(* CODESYS project PruebaReporte22.project

Project tree, tasks and I/O mapping:
  Device : CECC-LK, Festo AG & Co. KG, order no. 574418, version 3.5.3.1
    application Application
      libraries: Standard, * (System)
      task MainTask (cyclic, interval t#20ms, priority 20) calls PLC_PRG
      program PLC_PRG [LD]
      visualisation Visualization
    Onboard : CECC 14I/8O, Festo AG & Co. KG, version 3.4.5.5
        unmapped channels: Onboard Input, Onboard Output
      Digital Inputs
          unmapped channels: Onboard Input
      Digital Outputs
          unmapped channels: Onboard Output
  text list GlobalTextList
*)

// Device/Application/PLC_PRG
PROGRAM PLC_PRG
VAR
	S1: BOOL;
	B1: BOOL;
	Y1: BOOL;
	S2: BOOL;
	inicio: BOOL;
	Y3: BOOL;
	Y4: BOOL;
	Y2: BOOL;
	prevB1: BOOL;
	pulso: BOOL;
	fase: BOOL;
END_VAR
VAR // added by the converter: edge detectors and wires of the graphical bodies
    _w1, _w2, _w3 : BOOL;
END_VAR

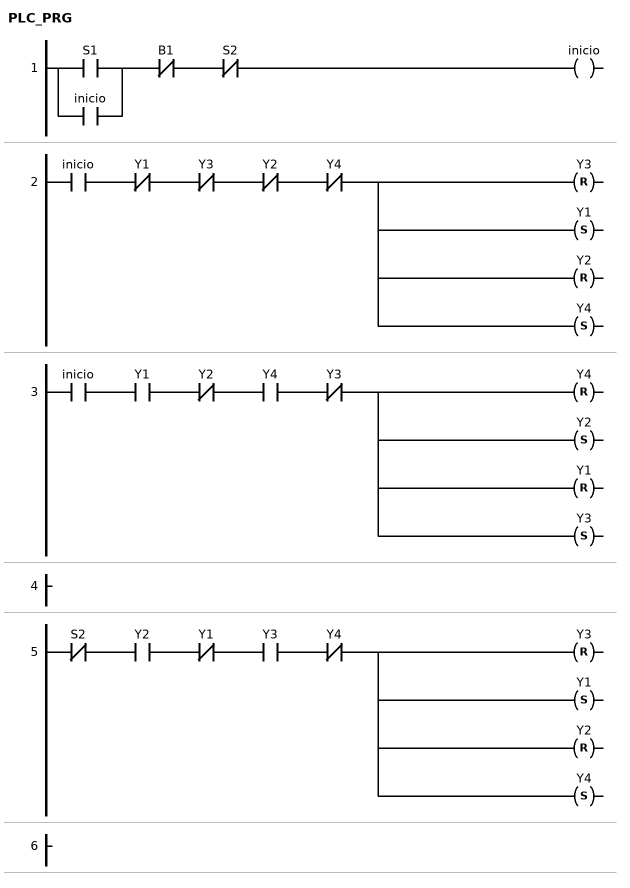
// NETWORK 1
inicio := (S1 OR inicio) AND NOT B1 AND NOT S2;

// NETWORK 2
_w1 := inicio AND NOT Y1 AND NOT Y3 AND NOT Y2 AND NOT Y4;
Y3 R= _w1;
Y1 S= _w1;
Y2 R= _w1;
Y4 S= _w1;

// NETWORK 3
_w2 := inicio AND Y1 AND NOT Y2 AND Y4 AND NOT Y3;
Y4 R= _w2;
Y2 S= _w2;
Y1 R= _w2;
Y3 S= _w2;

// NETWORK 4

// NETWORK 5
_w3 := NOT S2 AND Y2 AND NOT Y1 AND Y3 AND NOT Y4;
Y3 R= _w3;
Y1 S= _w3;
Y2 R= _w3;
Y4 S= _w3;

// NETWORK 6

END_PROGRAM

// Device/Application/Visualization
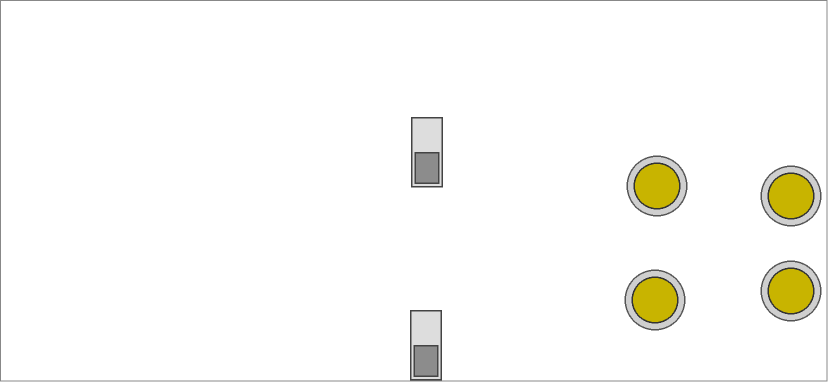
VISUALIZATION Visualization  // 828x382
    Lamp1 (622,151 70x70), variable: PLC_PRG.Y1, style: Lamp-Lamp1-Yellow
    DipSwitch (392,117 70x70), variable: PLC_PRG.S1, behaviour: TOGGLE, style: Switch-DipSwitch-Gray
    Lamp1 (756,161 70x70), variable: PLC_PRG.Y2, style: Lamp-Lamp1-Yellow
    DipSwitch (391,310 70x70), variable: PLC_PRG.S2, behaviour: TOGGLE, style: Switch-DipSwitch-Gray
    Lamp1 (620,265 70x70), variable: PLC_PRG.Y3, style: Lamp-Lamp1-Yellow
    Lamp1 (756,256 70x70), variable: PLC_PRG.Y4, style: Lamp-Lamp1-Yellow
END_VISUALIZATION
